FUNCTION_BLOCK BasicTestBlock2
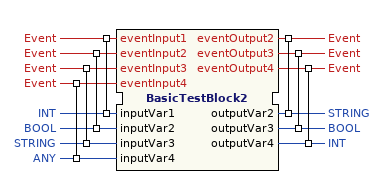
  EVENT_INPUT
    eventInput1 WITH inputVar1;
    eventInput2 WITH inputVar2;
    eventInput3 WITH inputVar3;
    eventInput4 WITH inputVar4;
  END_EVENT
  EVENT_OUTPUT
    eventOutput2 WITH outputVar2;
    eventOutput3 WITH outputVar3;
    eventOutput4 WITH outputVar4;
  END_EVENT
  VAR_INPUT
    inputVar1 : INT;
    inputVar2 : BOOL;
    inputVar3 : STRING;
    inputVar4 : ANY;
  END_VAR
  VAR_OUTPUT
    outputVar2 : STRING;
    outputVar3 : BOOL;
    outputVar4 : INT;
  END_VAR
  EC_STATES
    START;
  END_STATES
END_FUNCTION_BLOCK
